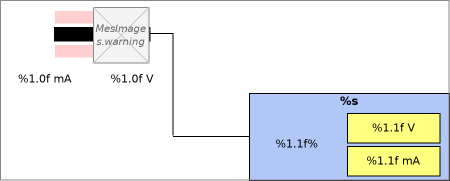
VISUALIZATION VISU_EFFLUVAGE  // 450x181
VAR_IN_OUT
	M_input_effluvage:	BLOCK_PRG_EFFLUVAGE;
END_VAR
    Line (140,33) (173,33)
    Line (173,136) (324,136)
    RoundedRectangle (55,11 93x12), invisible if: NOT M_input_effluvage.Effluvage.ALEFF.STATE_plasma
    Rectangle (2,64 86x30), "%1.0f mA", text variable: M_input_effluvage.Effluvage.ALEFF.STATE_current, invisible if: M_input_effluvage.Effluvage.ALEFF.STATE_OFF
    Rectangle (89,64 86x30), "%1.0f V", text variable: M_input_effluvage.Effluvage.ALEFF.STATE_tension, invisible if: M_input_effluvage.Effluvage.ALEFF.STATE_OFF
    RoundedRectangle (249,93 201x88), "%s", text list: 'TextList_Effluvage', text index: 1
    Textfield (257,132 80x24), "%1.1f%", text variable: M_input_effluvage.Effluvage.ALEFF.STATE_Setpoint_Power
    Rectangle (347,113 93x30), "%1.1f V", text variable: M_input_effluvage.Effluvage.PRM_Tension_attendue, invisible if: NOT M_input_effluvage.Effluvage.MANUAL, input disabled if: NOT PRG_USER.ACTU_USER.MAINTENANCE OR NOT PRG_EFFLUVAGE.Effluvage.Manual
        OnMouseClick: write the text variable via InputWithLimits, min 0, max M_input_effluvage.Effluvage.ALEFF.IN_CURRENT.CONF_Max
    RoundedRectangle (55,45 93x12), invisible if: NOT M_input_effluvage.Effluvage.ALEFF.STATE_plasma
    RoundedRectangle (54,27 96x14), colour toggle: PRG_EFFLUVAGE.Effluvage.ALEFF.STATE_ON, input disabled if: NOT PRG_USER.ACTU_USER.MAINTENANCE OR NOT PRG_EFFLUVAGE.Effluvage.Manual
        OnMouseClick: toggle M_input_effluvage.Effluvage.ALEFF.M_ON
    Image (93,7 56x56), invisible if: NOT M_input_effluvage.Effluvage.ALEFF.STATE_NOK, image: MesImages.warning
    Line (173,135) (173,33)
    Rectangle (347,146 93x30), "%1.1f mA", text variable: M_input_effluvage.Effluvage.PRM_consigne, invisible if: NOT M_input_effluvage.Effluvage.MANUAL, input disabled if: NOT PRG_USER.ACTU_USER.MAINTENANCE OR NOT PRG_EFFLUVAGE.Effluvage.Manual
        OnMouseClick: write the text variable via InputWithLimits, min 0, max M_input_effluvage.Effluvage.ALEFF.IN_CURRENT.CONF_Max
END_VISUALIZATION

(* stored: Version 1.1.0.1, ProductVersion 3.1.4024.10
   Visu VISU_EFFLUVAGE: Id {d11714ae-36ce-4bbb-85f5-ff4fd1cece99} *)
